FUNCTION_BLOCK EM_Can_Supply IMPLEMENTS ITF_Can_Supply, ITF_PackML
VAR
	fb_mem : STRUCT_EM_CanSupply;
	bFirstCycleExecuted : BOOL;
	
	//SubModules
	EM_Transport_Can_Supply1		: EM_Transport_Mechanische_Stop;
	EM_Transport_Can_Supply2		: EM_Transport;
	Sen_A1_Near						: CM_Sensor;
	Sen_A1_Far						: CM_Sensor;
	Sen_A2_Near						: CM_Sensor;
	Sen_A2_Far						: CM_Sensor;
	ValveDirection					: CM_Valve;  
END_VAR

(*
Tijn Verdurmen
*)//********************************Initiating***********************************
fb_mem.STS.State := PackML_StateMachine(State			:= fb_mem.STS.State,
										Start           := fb_mem.CS.Start,
										Stop            := fb_mem.CS.Stop,
										Reset           := fb_mem.CS.Reset,
										Abort           := fb_mem.CS.Abort,
										Clear           := fb_mem.CS.Clear,
										UnSuspend       := fb_mem.CS.UnSuspend,
										Suspend         := fb_mem.CS.Suspend,
										UnHold          := fb_mem.CS.UnHold,
										Hold            := fb_mem.CS.Hold,
										Starting_SC     := fb_mem.STS.Starting_SC,
										Execute_SC      := fb_mem.STS.Execute_SC,
										Completing_SC	:= fb_mem.STS.Completing_SC,
										Resetting_SC    := fb_mem.STS.Resetting_SC,
										Holding_SC      := fb_mem.STS.Holding_SC,
										Unholding_SC    := fb_mem.STS.Unholding_SC,
										Suspending_SC   := fb_mem.STS.Suspending_SC,
										Unsuspending_SC := fb_mem.STS.Unsuspending_SC,
										Aborting_SC     := fb_mem.STS.Aborting_SC,
										Clearing_SC     := fb_mem.STS.Clearing_SC,
										Stopping_SC     := fb_mem.STS.Stopping_SC);

//********************************Init***********************************
EM_Transport_Can_Supply1();
EM_Transport_Can_Supply2();			
										
//********************************ZEROING***********************************								
fb_mem.STS.Starting_SC 		:= FALSE;
fb_mem.STS.Execute_SC 		:= FALSE;
fb_mem.STS.Resetting_SC 	:= FALSE;
fb_mem.STS.Holding_SC 		:= FALSE;
fb_mem.STS.Unholding_SC 	:= FALSE;
fb_mem.STS.Suspending_SC 	:= FALSE;
fb_mem.STS.Unsuspending_SC 	:= FALSE;
fb_mem.STS.Aborting_SC 		:= FALSE;
fb_mem.STS.Clearing_SC 		:= FALSE;
fb_mem.STS.Stopping_SC 		:= FALSE;
fb_mem.STS.Completing_SC 	:= FALSE;

//********************************Auto manual logic***********************************
IF NOT bFirstCycleExecuted THEN
	EM_Transport_Can_Supply1.Auto();
	EM_Transport_Can_Supply2.Auto();
	ValveDirection.Auto := TRUE;
	bFirstCycleExecuted := TRUE;
END_IF

IF fb_mem.CS.Auto OR fb_mem.HMI.Auto THEN
	fb_mem.STS.Auto := TRUE;
	fb_mem.STS.Manueel := FALSE;
END_IF

IF fb_mem.CS.Manueel OR fb_mem.HMI.Manueel THEN
	fb_mem.STS.Auto := FALSE;
	fb_mem.STS.Manueel := TRUE;
END_IF

//********************Manupilatie***********8
IF fb_mem.SIM.Sen_A1_Near_TRUE THEN
	Sen_A1_Near.Output := TRUE;
END_IF
IF fb_mem.SIM.Sen_A1_Far_TRUE THEN
	Sen_A1_Far.Output := TRUE;
END_IF
IF fb_mem.SIM.Sen_A2_Near_TRUE THEN
	Sen_A2_Near.Output := TRUE;
END_IF
IF fb_mem.SIM.Sen_A2_Far_TRUE THEN
	Sen_A2_Far.Output := TRUE;
END_IF

//********************************Exeptionhandling***********************************

//********************************Action case***********************************
CASE fb_mem.STS.State OF
	E_State_PackML.IDLE 			: 
		//Do nothing
	E_State_PackML.STARTING 		:
		EM_Transport_Can_Supply1.Start();
		EM_Transport_Can_Supply2.Start();
		IF ((EM_Transport_Can_Supply1.State= E_State_PackML.EXECUTE) AND (EM_Transport_Can_Supply2.State= E_State_PackML.EXECUTE)) THEN
			ValveDirection.Close();	//=naar filler 1
				IF Sen_A1_Far.Output=TRUE AND Sen_A1_Near.Output=TRUE THEN //filler 2 hoeft nog niet vol te zijn om te starten
					ValveDirection.Open();	//=naar filler 2
					fb_mem.STS.Starting_SC := TRUE;
				END_IF
		END_IF
		
	E_State_PackML.EXECUTE		: // dit was execute
		//Hier heen en weer swichen totdat bijden buffers vol zijn en dus alle sensoren waar zijn met filler 1 prioriteit
		//Als Sen_A1_Far AND Sen_A1_Near AND !Sen_A2_Near THEN wissel naar A2 en vise versa
		IF Sen_A1_Far.Output=TRUE AND Sen_A2_Far.Output=TRUE AND Sen_A1_Near.Output=TRUE AND Sen_A2_Near.Output=FALSE THEN
			ValveDirection.Open();	//Richting_L naar filler 2 heet open
		END_IF
		IF Sen_A1_Far.Output=TRUE AND Sen_A2_Far.Output=TRUE AND Sen_A2_Near.Output=TRUE AND Sen_A1_Near.Output=FALSE THEN
			ValveDirection.Close();	//Richting_L naar filler 1
		END_IF
		IF Sen_A1_Far.Output=FALSE THEN
			ValveDirection.Close();		//Richting_L naar filler 1 heet close
		END_IF
	E_State_PackML.COMPLETING		:
		EM_Transport_Can_Supply1.Execute_SC();
		EM_Transport_Can_Supply2.Execute_SC();
		IF EM_Transport_Can_Supply1.State = E_State_PackML.COMPLETE AND EM_Transport_Can_Supply2.State = E_State_PackML.COMPLETE THEN
			fb_mem.STS.Completing_SC := TRUE;
		END_IF
	E_State_PackML.COMPLETE 		:
		fb_mem.STS.Completing_SC:=TRUE;
		
	E_State_PackML.RESETTING 		:
		EM_Transport_Can_Supply1.Reset();
		EM_Transport_Can_Supply2.Reset();
		IF	((EM_Transport_Can_Supply1.State= E_State_PackML.IDLE) AND (EM_Transport_Can_Supply2.State= E_State_PackML.IDLE)) THEN
			fb_mem.STS.Resetting_SC:=TRUE;
		END_IF
		
	E_State_PackML.HOLDING 			:
		EM_Transport_Can_Supply1.Hold();
		EM_Transport_Can_Supply2.Hold();
		IF	((EM_Transport_Can_Supply1.State= E_State_PackML.HELD) AND (EM_Transport_Can_Supply2.State= E_State_PackML.HELD)) THEN
			fb_mem.STS.Holding_SC:=TRUE;
		END_IF
		
	E_State_PackML.HELD 			:
		// Do nothing
	E_State_PackML.UNHOLDING 		:
		EM_Transport_Can_Supply1.Unhold();
		EM_Transport_Can_Supply2.Unhold();
		IF	((EM_Transport_Can_Supply1.State= E_State_PackML.EXECUTE) AND (EM_Transport_Can_Supply2.State= E_State_PackML.EXECUTE)) THEN
			fb_mem.STS.Unholding_SC:=TRUE;
		END_IF
		
	E_State_PackML.SUSPENDING 		:
		EM_Transport_Can_Supply1.Suspend();
		EM_Transport_Can_Supply2.Suspend();
		IF	((EM_Transport_Can_Supply1.State= E_State_PackML.SUSPENDED) AND (EM_Transport_Can_Supply2.State= E_State_PackML.SUSPENDED)) THEN
			fb_mem.STS.Suspending_SC:=TRUE;
		END_IF
		
	E_State_PackML.SUSPENDED 		:
		// Do nothing
		
	E_State_PackML.UNSUSPENDING 	:
		EM_Transport_Can_Supply1.Unsuspend();
		EM_Transport_Can_Supply2.Unsuspend();
		IF	((EM_Transport_Can_Supply1.State= E_State_PackML.EXECUTE) AND (EM_Transport_Can_Supply2.State= E_State_PackML.EXECUTE)) THEN
			fb_mem.STS.Unsuspending_SC:=TRUE;
		END_IF
	
	E_State_PackML.ABORTING			:
		EM_Transport_Can_Supply1.Abort();
		EM_Transport_Can_Supply2.Abort();
		IF	((EM_Transport_Can_Supply1.State= E_State_PackML.ABORTED) AND (EM_Transport_Can_Supply2.State= E_State_PackML.ABORTED)) THEN
			fb_mem.STS.Aborting_SC:=TRUE;
		END_IF
		
	E_State_PackML.ABORTED			:
		// Do nothing
		
	E_State_PackML.CLEARING 		:
		EM_Transport_Can_Supply1.Clear();
		EM_Transport_Can_Supply2.Clear();
		IF	((EM_Transport_Can_Supply1.State= E_State_PackML.STOPPED) AND (EM_Transport_Can_Supply2.State= E_State_PackML.STOPPED)) THEN
			fb_mem.STS.Clearing_SC:=TRUE;
		END_IF
		
	E_State_PackML.STOPPED			:
		// DO nothing
END_CASE 
//********************************HMI_Connection***********************************
fb_mem.STS.StringState     := TO_STRING(fb_mem.STS.State); 

//********************************ZEROING***********************************

fb_mem.CS.Auto            := FALSE;
fb_mem.CS.Manueel         := FALSE;
fb_mem.CS.Start           := FALSE;
fb_mem.CS.Stop            := FALSE;
fb_mem.CS.Reset           := FALSE;
fb_mem.CS.Abort           := FALSE;
fb_mem.CS.Clear           := FALSE;
fb_mem.CS.UnSuspend       := FALSE;
fb_mem.CS.Suspend         := FALSE;
fb_mem.CS.UnHold          := FALSE;
fb_mem.CS.Hold            := FALSE;

{warning 'add method implementation '}
METHOD Abort : BOOL
fb_mem.CS.Abort := TRUE;
END_METHOD

METHOD Aborting_SC : BOOL
VAR_INPUT
END_VAR
fb_mem.STS.Aborting_SC := TRUE;
END_METHOD

{warning 'add method implementation '}
METHOD Auto : BOOL
fb_mem.CS.Auto := TRUE;
Auto := fb_mem.STS.Auto;
END_METHOD

{warning 'add method implementation '}
METHOD Clear : BOOL
fb_mem.CS.Clear := TRUE;
END_METHOD

METHOD Clearing_SC : BOOL
VAR_INPUT
END_VAR
fb_mem.STS.Clearing_SC := TRUE;
END_METHOD

METHOD Completing_SC : BOOL
VAR_INPUT
END_VAR
fb_mem.STS.Completing_SC := TRUE;
END_METHOD

METHOD Execute_SC : BOOL
VAR_INPUT
END_VAR
fb_mem.STS.Execute_SC := TRUE;
END_METHOD

{warning 'add method implementation '}
METHOD FB_init : BOOL
VAR_INPUT
	bInitRetains : BOOL; // if TRUE, the retain variables are initialized (warm start / cold start)
	bInCopyCode : BOOL;  // if TRUE, the instance afterwards gets moved into the copy code (online change)
END_VAR
END_METHOD

{warning 'add method implementation '}
METHOD Hold : BOOL
fb_mem.CS.Hold := TRUE;
END_METHOD

METHOD Holding_SC : BOOL
VAR_INPUT
END_VAR
fb_mem.STS.Holding_SC := TRUE;
END_METHOD

{warning 'add method implementation '}
METHOD Manueel : BOOL
fb_mem.CS.Manueel := TRUE;
Manueel := fb_mem.STS.Manueel;
END_METHOD

{warning 'add method implementation '}
METHOD Reset : BOOL
fb_mem.CS.Reset := TRUE;
END_METHOD

METHOD Resetting_SC : BOOL
VAR_INPUT
END_VAR
fb_mem.STS.Resetting_SC := TRUE;
END_METHOD

{warning 'add method implementation '}
METHOD Start : BOOL
fb_mem.CS.Start := TRUE;
END_METHOD

METHOD Starting_SC : BOOL
VAR_INPUT
END_VAR
fb_mem.STS.Starting_SC := TRUE;
END_METHOD

{warning 'add property implementation'}
PROPERTY State : E_State_PackML
GET
State := fb_mem.STS.State;
END_GET
END_PROPERTY

{warning 'add method implementation '}
METHOD Stop : BOOL
fb_mem.CS.Stop := TRUE;
END_METHOD

METHOD Stopping_SC : BOOL
VAR_INPUT
END_VAR
fb_mem.STS.Stopping_SC := TRUE;
END_METHOD

{warning 'add method implementation '}
METHOD Suspend : BOOL
fb_mem.CS.Suspend := TRUE;
END_METHOD

METHOD Suspending_SC : BOOL
VAR_INPUT
END_VAR
fb_mem.STS.Suspending_SC := TRUE;
END_METHOD

{warning 'add method implementation '}
METHOD Unhold : BOOL
fb_mem.CS.Unhold := TRUE;
END_METHOD

METHOD Unholding_SC : BOOL
VAR_INPUT
END_VAR
fb_mem.STS.Unholding_SC := TRUE;
END_METHOD

{warning 'add method implementation '}
METHOD Unsuspend : BOOL
fb_mem.CS.Unsuspend := TRUE;
END_METHOD

METHOD Unsuspending_SC : BOOL
VAR_INPUT
END_VAR
fb_mem.STS.Unsuspending_SC := TRUE;
END_METHOD

{warning 'add method implementation '}
METHOD ZeroAllVar : BOOL
END_METHOD

END_FUNCTION_BLOCK

(* stored: Version 1.1.0.1, ProductVersion 3.1.4024.12
   POU EM_Can_Supply: Id {7d4cdf28-8942-4185-a3d0-da5253260d95}, SpecialFunc None
   Folder Methods: Id {36205fe7-9974-4236-80c4-92d328922c64}
   Folder Properties: Id {29891b51-a7e8-4e37-9797-88f55053a09e}
   Method Abort: Id {9ae06616-8598-42a0-a706-eabe119538d6}
   Method Aborting_SC: Id {1de7a9c8-59b9-42aa-b349-ad3bb6dba403}
   Method Auto: Id {3de32530-42eb-4924-90cf-af6c4db39c4e}
   Method Clear: Id {317eb4c1-dd26-4fc3-9ad1-01bb1f98d886}
   Method Clearing_SC: Id {9f05a99f-624c-465e-878e-f54db4026129}
   Method Completing_SC: Id {1bcf9784-5bcd-43d9-b48f-31129e0533dd}
   Method Execute_SC: Id {a4a0b4b3-25aa-4f68-970d-7630a42aa23c}
   Method FB_init: Id {bb9eb240-1942-4bca-86a2-4f174f21d3cc}
   Method Hold: Id {f1dd1fe1-f3d7-40f0-906a-c8d6bab2c883}
   Method Holding_SC: Id {ed8ba53c-b781-41b4-9526-4e77bb94145f}
   Method Manueel: Id {ef0b7851-5c06-402a-b160-6a9f79924c73}
   Method Reset: Id {b6d002df-90b6-47e2-a808-48474815356a}
   Method Resetting_SC: Id {e0ed2391-3347-4ca3-9de7-30a202fe8c62}
   Method Start: Id {48ae3542-0f2e-415e-bb40-f811f8674eae}
   Method Starting_SC: Id {d323944a-b0ac-4433-907c-bf2daacc2c6a}
   Property State: Id {5dfc3d61-b4c4-46e3-a627-12cb6b267db1}
   Get Get: Id {561168c5-4601-4861-9408-f30e5dbf64b3}
   Method Stop: Id {a34b6112-22b7-461a-8f9c-ac2ad867328a}
   Method Stopping_SC: Id {a3ee1337-f2e7-4ce8-96b8-edb70c657eb8}
   Method Suspend: Id {e31fc0d0-8941-4f6e-bd23-ea0b85ff8a3d}
   Method Suspending_SC: Id {057a2c9a-35d8-4727-9d42-6f8d08151c2d}
   Method Unhold: Id {0bcff60c-456a-411a-861d-f3bcd39f68ec}
   Method Unholding_SC: Id {24ddc2c1-1d2f-4964-b739-aa1adba8765a}
   Method Unsuspend: Id {6e53f95b-74e8-4513-965f-fc7292f6cb78}
   Method Unsuspending_SC: Id {95bfa227-be7a-4f57-a533-60914ada5233}
   Method ZeroAllVar: Id {f2032694-e612-411b-a380-5f4a137e6087} *)
